# EPICS substitutions: mc09/tpmacApp/Db/autohome.substitutions
file "$(EPICS_BASE)/db/autohome.db"
{

pattern
{SYS,              DEV,                 PLC,  PORT  }
{"XF:23ID1-BI",  "{Diag:5-Ax:Y}",      8     P0    }
{"XF:23ID1-BI",  "{Cam:Diag6-Ax:Y}",      9     P0    }
{"XF:23ID1-BI",  "{Cam:Diag6-Ax:Z}",      10    P0    }
{"XF:23ID1-BI",  "{Cam:Diag6-Ax:Zm}",      11    P0    }
{"XF:23ID1-BI",  "{Cam:Diag6-Ax:Foc}",      12    P0    }
}
